DATA_BLOCK "dbArchiveControlConveyor"
{ S7_Optimized_Access := 'TRUE' }
VERSION : 0.8
NON_RETAIN
"fbArchiveControlConveyor"

BEGIN

END_DATA_BLOCK

